// TIA Portal V20 export
// export: Created 2025-12-01T14:56:12.2218433Z, ExportSetting None, DisplayName Totally Integrated Automation Portal, DisplayVersion V20 Update 3, DisplayName TIA Portal Openness, DisplayVersion V20 Update 3, DisplayName TIA Portal Version Control Interface, DisplayVersion V20 Update 3, DisplayName STEP 7 Professional, DisplayVersion V20 Update 3, DisplayName STEP 7 Safety, DisplayVersion V20 Update 2, DisplayName WinCC Basic/Comfort/Advanced, DisplayVersion V20 Update 3, DisplayName WinCC Professional, DisplayVersion V20 Update 3, DisplayName WinCC Unified, DisplayVersion V20 Update 3
TYPE "UDT_SalidasExterioresDeMesa"
   STRUCT
      Avanzar_E1E3 : Bool;
      Retroceder_E1E3 : Bool;
      VelocidadLenta_E1E3 : Bool;
      Parar_E1E3 : Bool;
      Avanzar_E2E4 : Bool;
      Retroceder_E2E4 : Bool;
      VelocidadLenta_E2E4 : Bool;
      Parar_E2E4 : Bool;
      Ir_Pos_E1E3 : Bool;
      Ir_Pos_E2E4 : Bool;
      Subir_MElevadora : Bool;   // utilizar para maqueta FS
      Bajar_MElevadora : Bool;   // utilizar para maqueta FS
      Subir_TP_E1E3 : Bool;
      Bajar_TP_E1E3 : Bool;
      Subir_TP_E2E4 : Bool;
      Bajar_TP_E2E4 : Bool;
      Subir_TP_E3E1 : Bool;
      Bajar_TP_E3E1 : Bool;
      Subir_TP_E4E2 : Bool;
      Bajar_TP_E4E2 : Bool;
      PickUpOK : Bool;   // CS y FS
      DepositOK : Bool;   // CS y FS
      LoadOK : Bool;
      UnLoadOK : Bool;
      UnLoadComplete : Bool;
      Ir_Pos_S2_Cil1 : Bool;   // Utilizar para empujador extendido
      Ir_Pos_S3_Cil1 : Bool;   // Utilizar para empujador recogido
      Ir_Pos_S4_Cil1 : Bool;
      Ir_Pos_S2_Cil2 : Bool;
      Ir_Pos_S3_Cil2 : Bool;
      Ir_Pos_S4_Cil2 : Bool;
      Avanzar_Entrada : Bool;
      Avanzar_Salida : Bool;
      Ir_Pos_S2 : Bool;
      Ir_Pos_S4 : Bool;
      Disparo_SCR : Bool;
      HB_PTF_FIN { ExternalAccessible := 'False'; ExternalVisible := 'False'; ExternalWritable := 'False'} : Bool;
      HB_ATF_INI { ExternalAccessible := 'False'; ExternalVisible := 'False'; ExternalWritable := 'False'} : Bool;
      HB_PARO_Zona { ExternalAccessible := 'False'; ExternalVisible := 'False'; ExternalWritable := 'False'} : Bool;
   END_STRUCT;
END_TYPE
